// TwinCAT 3 PLC project Motion_Test_Stand
// ProgramVersion: 3.1.4022.7
// libraries:
//   LCLS General, * (SLAC)
//   lcls-twincat-motion, * (SLAC)
//   PMPS, * (SLAC - LCLS)
//   Tc2_Standard, * (Beckhoff Automation GmbH)
//   Tc2_System, * (Beckhoff Automation GmbH)
//   Tc3_Module, * (Beckhoff Automation GmbH)
// project tree:
//   DUTs/ ST_EPSLimits.TcDUT
//   GVLs/ GVL_EPS.TcGVL
//   / PlcTask.TcTTO (not stored)
//   POUs/ FB_CheckEPS.TcPOU, F_InRange.TcPOU, MAIN.TcPOU
// real-time tasks:
//   TASK PlcTask: cycle T#10ms, priority 20, ADS port 350
// motion (NC):
// I/O:
//   DEVICE Device 1 (EtherCAT), AmsNetId 172.21.148.87.2.1
//     Term 1 (EK1200)
// variable links:
//   Motion_Test_Stand Instance <-> Device 1 (EtherCAT)/Term 1 (EK1200)/M1-EL1084
//     PlcTask Inputs/MAIN.bLimitBackwardEnable <-> Channel 1/Input
//     PlcTask Inputs/MAIN.bLimitForwardEnable <-> Channel 2/Input
//   Motion_Test_Stand Instance <-> Device 1 (EtherCAT)/Term 1 (EK1200)/M1-EL5042
//     PlcTask Inputs/MAIN.M1.nRawEncoderULINT <-> FB Inputs Channel 1/Position
//   Motion_Test_Stand Instance <-> NC-Task 1 SAF/Axes/Axis 1
//     PlcTask Inputs/MAIN.M1.Axis.NcToPlc <-> Outputs/ToPlc
//     PlcTask Outputs/MAIN.M1.Axis.PlcToNc <-> Inputs/FromPlc

// ---- DUTs/ST_EPSLimits.TcDUT
TYPE ST_EPSLimits :
STRUCT
    {attribute 'pytmc' := '
        pv: FwdLimit
        io: io
    '}
    fFwd_Limits : REAL;
    {attribute 'pytmc' := '
        pv: BwdLimit
        io: io
    '}
    fBwd_Limits	: REAL;
    {attribute 'pytmc' := 'pv: ST'}
    stEPS 		: DUT_EPS;
END_STRUCT
END_TYPE

// ---- GVLs/GVL_EPS.TcGVL
VAR_GLOBAL

{attribute 'pytmc' := 'pv: TST:MOTION:EPS_ARRAY'}
aEPS_TEST : ARRAY [1 .. 2] OF ST_EPSLimits;
END_VAR

// ---- POUs/FB_CheckEPS.TcPOU
FUNCTION_BLOCK FB_CheckEPS
VAR_IN_OUT
	// Motor that will stop on plc limits
    stMotor	: ST_MotionStage;
	// Array of plc limits and states
    aEPSLimits : ARRAY [*] OF ST_EPSLimits;
END_VAR
VAR_INPUT
	// Encoder Position, Current position of motor. Needed for the case where the motor and encoders are seperate.
	fPosition : REAL;
END_VAR
VAR_OUTPUT
END_VAR
VAR
	nPreviousState : DINT;
	nIndex: DINT;
    nEPSIndex: DINT;
    fbBwdEPS: FB_EPS;
    fbFwdEPS: FB_EPS;
END_VAR

fbBwdEps(eps:=stMotor.stEPSBackwardEnable);
fbFwdEPS(eps:=stMotor.stEPSForwardEnable);

// Look through possible states to see witch state we are in
FOR nIndex := LOWER_BOUND(aEPSLimits, 1) TO UPPER_BOUND(aEPSLimits, 1) BY 1 DO
    IF aEPSLimits[nIndex].stEPS.bEPS_OK THEN
        nEPSIndex := nIndex;
		EXIT; // Stop Looking
    END_IF
END_FOR

IF (NOT (nPreviousState = nEPSIndex)) THEN
	// Clear Previous State Errors
	stMotor.stEPSBackwardEnable.nFlags := 16#FFFFFFFF;
	stMotor.stEPSBackwardEnable.bEPS_OK := TRUE;
	stMotor.stEPSForwardEnable.nFlags := 16#FFFFFFFF;
	stMotor.stEPSForwardEnable.bEPS_OK := TRUE;
END_IF

// Check if position is in plc limit rage
IF fPosition > aEPSLimits[nEPSIndex].fBwd_Limits THEN
	// Winith Limits
    fbBwdEPS.setBit(DINT_TO_BYTE(nEPSIndex), TRUE);
ELSE
	// Outside Limits
    fbBwdEPS.setBit(DINT_TO_BYTE(nEPSIndex), FALSE);
END_IF

IF fPosition < aEPSLimits[nEPSIndex].fFwd_Limits THEN
    fbFwdEPS.setBit(DINT_TO_BYTE(nEPSIndex), TRUE);
ELSE
    fbFwdEPS.setBit(DINT_TO_BYTE(nEPSIndex), FALSE);
END_IF

nPreviousState := nEPSIndex; // Update Previous State

END_FUNCTION_BLOCK

// ---- POUs/F_InRange.TcPOU
FUNCTION F_InRange : BOOL
VAR_INPUT
    value 		: LREAL;
    lower_limit : LREAL;
    upper_limit : LREAL;
END_VAR
VAR
END_VAR

F_InRange := (lower_limit < value) AND (value < upper_limit);

END_FUNCTION

// ---- POUs/MAIN.TcPOU
PROGRAM MAIN
VAR

{attribute 'pytmc' := 'pv: TST:MOTION'}
{attribute 'TcLinkTo' := '.nRawEncoderULINT     := TIID^Device 1 (EtherCAT)^Term 1 (EK1200)^M1-EL5042^FB Inputs Channel 1^Position'}
M1: ST_MotionStage := (sName := 'TST:MOTION',
                        bPowerSelf := True,
                        nEnableMode:= ENUM_StageEnableMode.DURING_MOTION);

{attribute 'TcLinkTo' := 'TIID^Device 1 (EtherCAT)^Term 1 (EK1200)^M1-EL1084^Channel 1^Input'}
bLimitBackwardEnable AT %I* : BOOL;

{attribute 'TcLinkTo' := 'TIID^Device 1 (EtherCAT)^Term 1 (EK1200)^M1-EL1084^Channel 2^Input'}
bLimitForwardEnable AT %I* : BOOL;

fbmotion1 : FB_MotionStage;

	fbEPS : FB_EPS;
	bInit : BOOL := TRUE;
	nIndex : UINT := 1;
	nEPSIndex : UINT := 1;
	fPos : LREAL;
	
	{attribute 'pytmc' := 'pv: TST:MOTION:EPS_TST_TOGGLE'}
	btest1	: BOOL := TRUE;
	
	bEPS_OK : BOOL;
	bInRange : BOOL;

	fbEPS_States : FB_CheckEPS;
END_VAR

// GX-F8A are NPN 
M1.bLimitForwardEnable 	:= Not bLimitForwardEnable;
M1.bLimitBackwardEnable := Not bLimitBackwardEnable;

M1.bHardwareEnable := True;
fbmotion1(stMotionStage:=M1);

IF bInit THEN
	aEPS_TEST[1].fBwd_Limits := -0.5;
	aEPS_TEST[1].fFwd_Limits := 0.5;
	
	aEPS_TEST[2].fBwd_Limits := -2;
	aEPS_TEST[2].fFwd_Limits := 2;
	
	
	bInit := FALSE;
END_IF

fPos := M1.stAxisStatus.fActPosition;

fbEPS(eps:= aEPS_TEST[1].stEPS);
fbEPS.setDescription('TST_TOGGLE: TRUE;IN LIMITS; NOT TEST 2');
fbEPS.setBit(0, btest1);
fbEPS.setBit(1, F_InRange(fPos, aEPS_TEST[1].fBwd_Limits, aEPS_TEST[1].fFwd_Limits));
fbEPS.setBit(2, NOT aEPS_TEST[2].stEPS.bEPS_OK);

fbEPS(eps:= aEPS_TEST[2].stEPS);
fbEPS.setDescription('TST_TOGGLE: FALSE;IN LIMITS; NOT TEST 1');
fbEPS.setBit(0, NOT btest1);
fbEPS.setBit(1, F_InRange(fPos, aEPS_TEST[2].fBwd_Limits, aEPS_TEST[2].fFwd_Limits));
fbEPS.setBit(2, NOT aEPS_TEST[1].stEPS.bEPS_OK);


bInRange := F_InRange(fPos, aEPS_TEST[nEPSIndex].fBwd_Limits, aEPS_TEST[nEPSIndex].fFwd_Limits);

fbEPS_States(stMotor:=M1, fPosition:=M1.stAxisStatus.fActPosition, aEPSLimits:=aEPS_TEST);

END_PROGRAM
